INTERFACE I_Mc2MotionJogTask EXTENDS I_Mc2MotionTask

PROPERTY JogBackwards : BOOL
SET
END_SET
END_PROPERTY

PROPERTY JogForward : BOOL
SET
END_SET
END_PROPERTY

PROPERTY Mode : E_JogMode
SET
END_SET
END_PROPERTY

PROPERTY Position : LREAL
SET
END_SET
END_PROPERTY

END_INTERFACE

(* stored: Version 1.1.0.1, ProductVersion 3.1.4026.20
   Itf I_Mc2MotionJogTask: Id {e8e42b92-1ac7-4dad-958f-f15ca9216c49}
   Property JogBackwards: Id {08ee9f05-8c8f-4237-b54e-4bdbfdf91a60}
   Set Set: Id {f406ce6f-55fe-4cd6-8718-e969becf6ad1}
   Property JogForward: Id {d7e1f925-cf09-4f09-8ec7-596affe82a44}
   Set Set: Id {c5ffd81f-04a0-4bbe-9671-4c2c805e41ca}
   Property Mode: Id {521aea47-3e4b-4b0e-b834-6e6fd99cc11d}
   Set Set: Id {08520522-9237-4857-af3c-b7eb9f5117e7}
   Property Position: Id {58db24ae-f50c-442a-be74-d8cd20b28d38}
   Set Set: Id {4ae7819d-a48d-495d-8828-0f07e1484982} *)
